TEXTLIST TextListGlobal
  0 = 'Aktualny stan : ' | pl: 'Aktualny stan : ' | en: 'Current state : ' | de: 'Aktueller Zustand : '
  1 = 'Aktualny tryb : ' | pl: 'Aktualny tryb : ' | en: 'Current mode : ' | de: 'Aktueller Modus : '
  2 = 'Anuluj' | pl: 'Anuluj' | en: 'Cancel' | de: 'Stornieren'
  3 = 'Przywróc domyślną wartość' | pl: 'Przywróc domyślną wartość' | en: 'Restore default value' | de: 'Standardwert wiederherstellen'
  4 = 'Zapisz' | pl: 'Zapisz' | en: 'Save' | de: 'Speichern'
  5 = 'Wartość domyślna' | pl: 'Wartość domyślna' | en: 'Default value' | de: 'Standardwert'
  6 = 'Wartość' | pl: 'Wartość' | en: 'Value' | de: 'Wert'
  7 = 'Brak wybranej receptury' | pl: 'Brak wybranej receptury' | en: 'No recipe selected' | de: 'Kein Rezept ausgewählt'
   = ''
END_TEXTLIST

(* stored: Version 1.1.0.1
   TextList TextListGlobal: Id {9d88ac8d-dfee-05e3-3c03-115625ce9742} *)
